// TIA Portal V18 export
DATA_BLOCK "SS1_CPU1215_DO_Vars"   // DB11014
{ S7_Optimized_Access := 'FALSE' }
VERSION : 0.1
// stored: AutoNumber false, DBAccessibleFromOPCUA true, IsOnlyStoredInLoadMemory false, IsWriteProtectedInAS false
   VAR
      DO1 { S7_SetPoint := 'True'} : "UDT_DOadv";
      DO2 { S7_SetPoint := 'True'} : "UDT_DOadv";
      DO3 { S7_SetPoint := 'True'} : "UDT_DOadv";
      DO4 { S7_SetPoint := 'True'} : "UDT_DOadv";
      DO5 { S7_SetPoint := 'True'} : "UDT_DOadv";
      DO6 : "UDT_DOadv";
      DO7 { S7_SetPoint := 'True'} : "UDT_DOadv";
      DO8 { S7_SetPoint := 'True'} : "UDT_DOadv";
      DO9 { S7_SetPoint := 'True'} : "UDT_DOadv";
      DO10 { S7_SetPoint := 'True'} : "UDT_DOadv";
   END_VAR
BEGIN
END_DATA_BLOCK
